{attribute 'qualified_only'}
VAR_GLOBAL CONSTANT
    stClamping : ST_ClampingSafetyConfig := (fMinimumAllowedPosition := 21.0, fModeSwitchVelocityMax := 0.01, bEnableHardMaxClampTorqueCheck := FALSE, fHardMaxClampTorquePercent := 0.0);
    stStop : ST_StopSafetyConfig := (tTimeout := T#10S);
    stStartup : ST_StartupSafetyConfig := (tEnableTimeout := T#15S);
END_VAR

(* stored: Version 1.1.0.1, ProductVersion 3.1.4026.20
   GVL GVL_SafetyConfig: Id {1914259c-8fe9-49d7-820e-667631cb12b8} *)
